Staubli VAL3: Circle3point.pgx

public program Circle3point(pointRx& x_pPointCenter, num& x_nDia, tool x_tTool, bool& x_bOK)
  local num l_ni
  local num x1
  local num x2
  local num x3
  local num y1
  local num y2
  local num y3
  local num l_nError
  local point l_pPoint[3]
  local point l_pCenter
  local frame l_fFrame
  local num l_nErr
begin
  //三点法-圆
  nFrame1Err=setFrame(pFrameRefPt[0],pFrameRefPt[1],pFrameRefPt[2],fFrame1)
  if nFrame1Err==-1
    popUpMsg("X方向点离原点太近")
  endIf
  if nFrame1Err==-2
    popUpMsg("Y方向点离原点太近")
  endIf
  //  l_nErr=setFrame(x_pt[0],x_pt[1],x_pt[2],fFrame)
  if nFrame1Err==0
    l_pCenter=here(x_tTool,fFrame1)
    l_pCenter.trsf=position(pFrameRefPt[0],fFrame1)
    for l_ni=0 to 2 step 1
      l_pPoint[l_ni].trsf=position(pFrameRefPt[l_ni],fFrame1)
    endFor
    x1=l_pPoint[0].trsf.x
    x2=l_pPoint[1].trsf.x
    x3=l_pPoint[2].trsf.x
    y1=l_pPoint[0].trsf.y
    y2=l_pPoint[1].trsf.y
    y3=l_pPoint[2].trsf.y
    if ((x3-x1)*(y2-y1)-(x2-x1)*(y3-y1))!=0
      l_pCenter.trsf.x=((y2-y1)*(y3*y3-y1*y1+x3*x3-x1*x1)-(y3-y1)*(y2*y2-y1*y1+x2*x2-x1*x1))/(2*(x3-x1)*(y2-y1)-2*(x2-x1)*(y3-y1))
      l_pCenter.trsf.y=((x2-x1)*(x3*x3-x1*x1+y3*y3-y1*y1)-(x3-x1)*(x2*x2-x1*x1+y2*y2-y1*y1))/(2*(y3-y1)*(x2-x1)-2*(y2-y1)*(x3-x1))
      x_pPointCenter.trsf=position(l_pCenter,world)
      //修改
      x_pPointCenter.trsf.rx=fFrame1.trsf.rx
      x_pPointCenter.trsf.ry=fFrame1.trsf.ry
      x_pPointCenter.trsf.rz=fFrame1.trsf.rz
      //
      x_nDia=2*sqrt((l_pPoint[0].trsf.x-l_pCenter.trsf.x)*(l_pPoint[0].trsf.x-l_pCenter.trsf.x)+(l_pPoint[0].trsf.y-l_pCenter.trsf.y)*(l_pPoint[0].trsf.y-l_pCenter.trsf.y))
      x_bOK=true
    else
      x_bOK=false
      x_nDia=0
    endIf
  else
    x_bOK=false
    x_nDia=0
  endIf
end
